# EPICS substitutions: db/MLRun.substitutions
file "/epics/iocs/MachineLearn/db/MLRun.db"
{
pattern
{C1,   C2,   C3  }
{"01", "11", "21"}
{"02", "12", "22"}
{"03", "13", "23"}
{"04", "14", "24"}
{"05", "15", "25"}
{"06", "16", "26"}
{"07", "17", "27"}
{"08", "18", "28"}
{"09", "19", "29"}
{"10", "20", "30"}
}
